PROGRAM motor_starter_control
VAR PERSISTENT
	//Example motor starter block.  
	u_3160 : motor_starter;

END_VAR

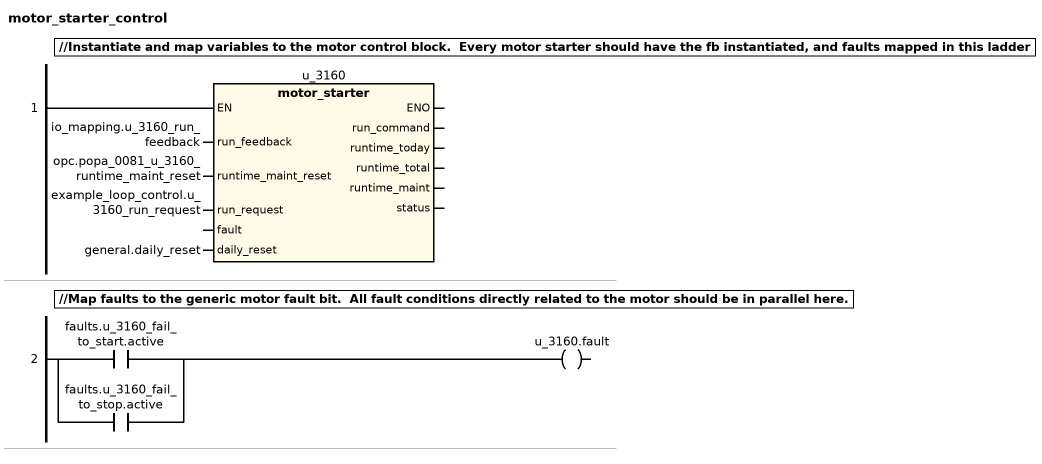
// NETWORK 1
// label: //Instantiate and map variables to the motor control block.  Every motor starter should have the fb instantiated, and faults mapped in this ladder
u_3160(
    run_feedback := io_mapping.u_3160_run_feedback,
    runtime_maint_reset := opc.popa_0081_u_3160_runtime_maint_reset,
    run_request := example_loop_control.u_3160_run_request,
    daily_reset := general.daily_reset); // motor_starter

// NETWORK 2
// label: //Map faults to the generic motor fault bit.  All fault conditions directly related to the motor should be in parallel here.
u_3160.fault := faults.u_3160_fail_to_start.active OR faults.u_3160_fail_to_stop.active;

END_PROGRAM

(* stored: Version 1.1.0.1, ProductVersion 3.1.4024.12
   POU motor_starter_control: Id {875228a8-8d81-4320-b913-8585bf7e4dcc}, SpecialFunc None *)
